% RSLogix 500 project DIGI_FILL_STATION.RSS, saved by version 8.30.00.16 %
PROJECT "UNTITLED"    % processor: Bul.1763 MicroLogix 1100 Series B %

PROGRAM FILES
  LAD 2 "MAIN"  3 rungs
  LAD 3 "I/O"  8 rungs
  LAD 4 "CONTROLS"  9 rungs

DATA FILES
  O0 OUTPUT  5 elements
  I1 INPUT  7 elements
  S2 STATUS  66 elements
  B3 BINARY  2 elements
  T4 TIMER  5 elements
  C5 COUNTER  1 elements
  R6 CONTROL  1 elements
  N7 INTEGER  1 elements
  F8 FLOAT  1 elements

LADDER 2 "MAIN"
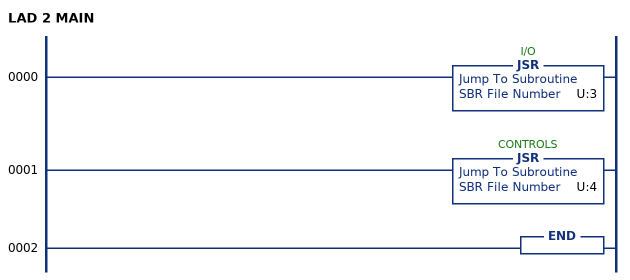
% Rung: 0 %
SOR JSR U:3 EOR
%   U:3  "I/O" %
% Rung: 1 %
SOR JSR U:4 EOR
%   U:4  "CONTROLS" %
% Rung: 2 %
SOR END EOR

LADDER 3 "I/O"
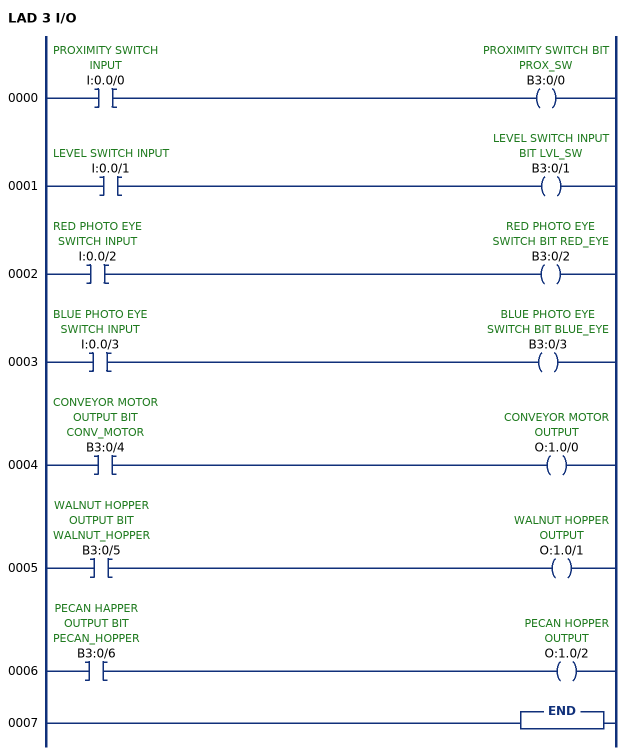
% Rung: 0 %
SOR XIC I:0.0/0 OTE B3:0/0 EOR
%   I:0.0/0  "PROXIMITY SWITCH INPUT" %
%   B3:0/0  PROX_SW  "PROXIMITY SWITCH BIT" %
% Rung: 1 %
SOR XIC I:0.0/1 OTE B3:0/1 EOR
%   I:0.0/1  "LEVEL SWITCH INPUT" %
%   B3:0/1  LVL_SW  "LEVEL SWITCH INPUT BIT" %
% Rung: 2 %
SOR XIC I:0.0/2 OTE B3:0/2 EOR
%   I:0.0/2  "RED PHOTO EYE SWITCH INPUT" %
%   B3:0/2  RED_EYE  "RED PHOTO EYE SWITCH BIT" %
% Rung: 3 %
SOR XIC I:0.0/3 OTE B3:0/3 EOR
%   I:0.0/3  "BLUE PHOTO EYE SWITCH INPUT" %
%   B3:0/3  BLUE_EYE  "BLUE PHOTO EYE SWITCH BIT" %
% Rung: 4 %
SOR XIC B3:0/4 OTE O:1.0/0 EOR
%   B3:0/4  CONV_MOTOR  "CONVEYOR MOTOR OUTPUT BIT" %
%   O:1.0/0  "CONVEYOR MOTOR OUTPUT" %
% Rung: 5 %
SOR XIC B3:0/5 OTE O:1.0/1 EOR
%   B3:0/5  WALNUT_HOPPER  "WALNUT HOPPER OUTPUT BIT" %
%   O:1.0/1  "WALNUT HOPPER OUTPUT" %
% Rung: 6 %
SOR XIC B3:0/6 OTE O:1.0/2 EOR
%   B3:0/6  PECAN_HOPPER  "PECAN HAPPER OUTPUT BIT" %
%   O:1.0/2  "PECAN HOPPER OUTPUT" %
% Rung: 7 %
SOR END EOR

LADDER 4 "CONTROLS"
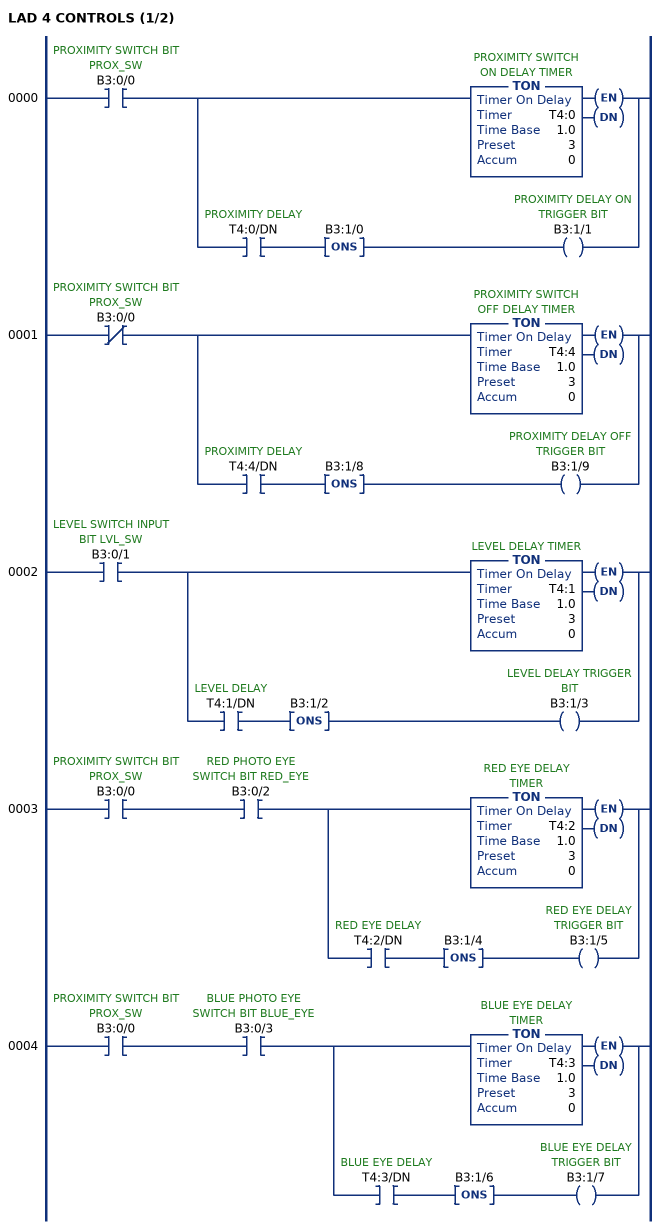
% Rung: 0 %
SOR XIC B3:0/0 BST TON T4:0 1.0 3 0 NXB XIC T4:0/DN ONS B3:1/0 OTE B3:1/1 BND EOR
%   B3:0/0  PROX_SW  "PROXIMITY SWITCH BIT" %
%   T4:0  "PROXIMITY SWITCH ON DELAY TIMER" %
%   T4:0/DN  "PROXIMITY DELAY" %
%   B3:1/1  "PROXIMITY DELAY ON TRIGGER BIT" %
% Rung: 1 %
SOR XIO B3:0/0 BST TON T4:4 1.0 3 0 NXB XIC T4:4/DN ONS B3:1/8 OTE B3:1/9 BND EOR
%   B3:0/0  PROX_SW  "PROXIMITY SWITCH BIT" %
%   T4:4  "PROXIMITY SWITCH OFF DELAY TIMER" %
%   T4:4/DN  "PROXIMITY DELAY" %
%   B3:1/9  "PROXIMITY DELAY OFF TRIGGER BIT" %
% Rung: 2 %
SOR XIC B3:0/1 BST TON T4:1 1.0 3 0 NXB XIC T4:1/DN ONS B3:1/2 OTE B3:1/3 BND EOR
%   B3:0/1  LVL_SW  "LEVEL SWITCH INPUT BIT" %
%   T4:1  "LEVEL DELAY TIMER" %
%   T4:1/DN  "LEVEL DELAY" %
%   B3:1/3  "LEVEL DELAY TRIGGER BIT" %
% Rung: 3 %
SOR XIC B3:0/0 XIC B3:0/2 BST TON T4:2 1.0 3 0 NXB XIC T4:2/DN ONS B3:1/4 OTE B3:1/5 BND EOR
%   B3:0/0  PROX_SW  "PROXIMITY SWITCH BIT" %
%   B3:0/2  RED_EYE  "RED PHOTO EYE SWITCH BIT" %
%   T4:2  "RED EYE DELAY TIMER" %
%   T4:2/DN  "RED EYE DELAY" %
%   B3:1/5  "RED EYE DELAY TRIGGER BIT" %
% Rung: 4 %
SOR XIC B3:0/0 XIC B3:0/3 BST TON T4:3 1.0 3 0 NXB XIC T4:3/DN ONS B3:1/6 OTE B3:1/7 BND EOR
%   B3:0/0  PROX_SW  "PROXIMITY SWITCH BIT" %
%   B3:0/3  BLUE_EYE  "BLUE PHOTO EYE SWITCH BIT" %
%   T4:3  "BLUE EYE DELAY TIMER" %
%   T4:3/DN  "BLUE EYE DELAY" %
%   B3:1/7  "BLUE EYE DELAY TRIGGER BIT" %

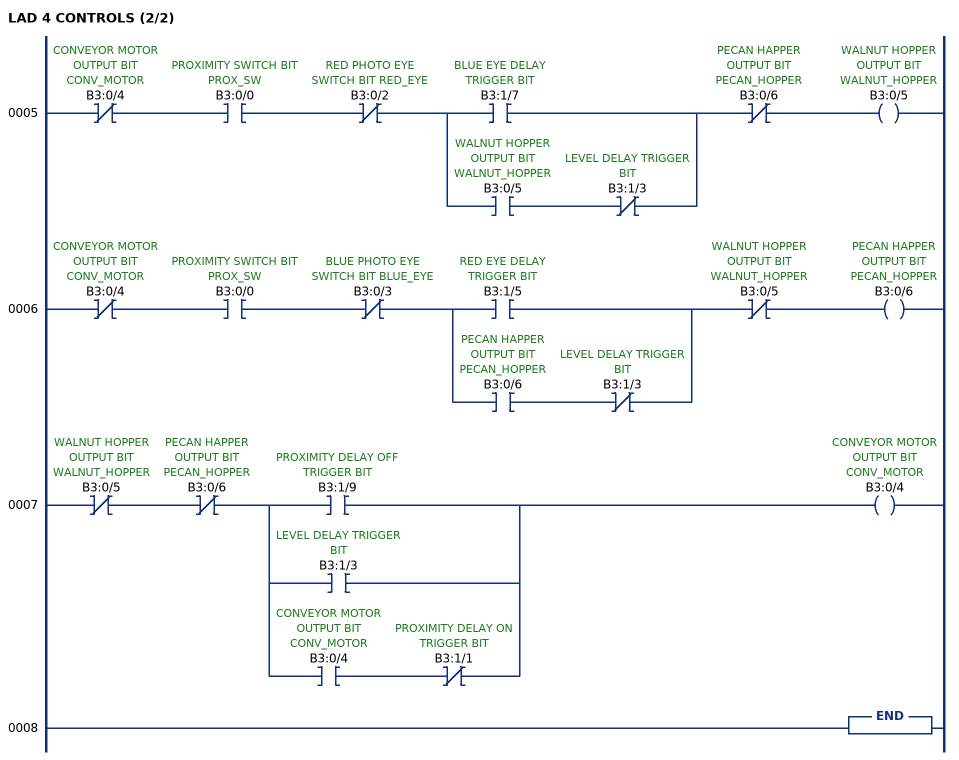
% Rung: 5 %
SOR XIO B3:0/4 XIC B3:0/0 XIO B3:0/2 BST XIC B3:1/7 NXB XIC B3:0/5 XIO B3:1/3 BND XIO B3:0/6 OTE B3:0/5 EOR
%   B3:0/4  CONV_MOTOR  "CONVEYOR MOTOR OUTPUT BIT" %
%   B3:0/0  PROX_SW  "PROXIMITY SWITCH BIT" %
%   B3:0/2  RED_EYE  "RED PHOTO EYE SWITCH BIT" %
%   B3:1/7  "BLUE EYE DELAY TRIGGER BIT" %
%   B3:0/5  WALNUT_HOPPER  "WALNUT HOPPER OUTPUT BIT" %
%   B3:1/3  "LEVEL DELAY TRIGGER BIT" %
%   B3:0/6  PECAN_HOPPER  "PECAN HAPPER OUTPUT BIT" %
% Rung: 6 %
SOR XIO B3:0/4 XIC B3:0/0 XIO B3:0/3 BST XIC B3:1/5 NXB XIC B3:0/6 XIO B3:1/3 BND XIO B3:0/5 OTE B3:0/6 EOR
%   B3:0/4  CONV_MOTOR  "CONVEYOR MOTOR OUTPUT BIT" %
%   B3:0/0  PROX_SW  "PROXIMITY SWITCH BIT" %
%   B3:0/3  BLUE_EYE  "BLUE PHOTO EYE SWITCH BIT" %
%   B3:1/5  "RED EYE DELAY TRIGGER BIT" %
%   B3:0/6  PECAN_HOPPER  "PECAN HAPPER OUTPUT BIT" %
%   B3:1/3  "LEVEL DELAY TRIGGER BIT" %
%   B3:0/5  WALNUT_HOPPER  "WALNUT HOPPER OUTPUT BIT" %
% Rung: 7 %
SOR XIO B3:0/5 XIO B3:0/6 BST XIC B3:1/9 NXB XIC B3:1/3 NXB XIC B3:0/4 XIO B3:1/1 BND OTE B3:0/4 EOR
%   B3:0/5  WALNUT_HOPPER  "WALNUT HOPPER OUTPUT BIT" %
%   B3:0/6  PECAN_HOPPER  "PECAN HAPPER OUTPUT BIT" %
%   B3:1/9  "PROXIMITY DELAY OFF TRIGGER BIT" %
%   B3:1/3  "LEVEL DELAY TRIGGER BIT" %
%   B3:0/4  CONV_MOTOR  "CONVEYOR MOTOR OUTPUT BIT" %
%   B3:1/1  "PROXIMITY DELAY ON TRIGGER BIT" %
% Rung: 8 %
SOR END EOR

DATA TABLE (non-zero values as saved)
DATA T4
% .PRE .ACC %
% T4:0 % 3 0
% T4:1 % 3 0
% T4:2 % 3 0
% T4:3 % 3 0
% T4:4 % 3 0
